Universal Robots PolyScope program: DEMO_ghost4.urp

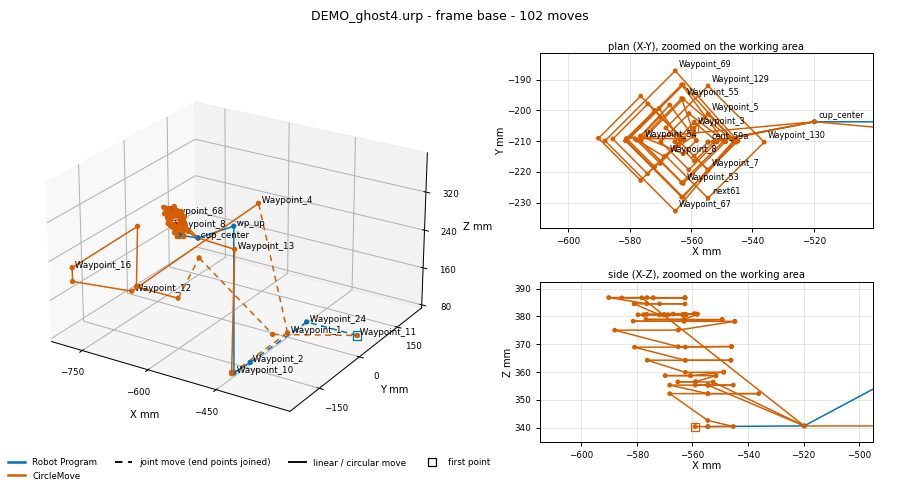
[picture p0: tool path of DEMO_ghost4.urp in frame base, 102 of 102 moves have a stored position in this frame; points joined in program order, loops and branches not executed]
Program DEMO_ghost4 (createdIn=3.3.3.292 lastSavedIn=3.3.3.292 directory=/programs/usbdisk_0 installation=default robotSerialNumber=2016353566)
Calibrated DH parameters: a=[0.000241, -0.028217, -0.285075, -0.000076, 0.000104, 0]; d=[0.089155, 574.834368, -342.811798, -231.912434, 0.094822, 0.082605]; alpha=[1.570306, 0.000738, 0.001161, 1.569845, -1.570892, 0]; deltaTheta=[0.000027, 1.504353, -0.747309, -0.757122, 0.000051, -0.000036]
Robot Program (runOnlyOnce=true motionType=MoveJ speed=1.047198 acceleration=1.396263 recalculateMotions=false)
  'c250g_w360g'
  URCap com.ur.urcap.OnRobot.HelloWorldNode data=depthCompensate = false
    | width = 40
    | name = RG2(40)
    | force = 40
  MoveJ speed 20 deg/s, acceleration 30 deg/s^2 (recalculateMotions=false)
    Waypoint Waypoint_11: TCP in base x=-315.829 y=31.141 z=99.108 mm, rx=0.0221 ry=-2.2156 rz=2.1951 rad; joints [-58.8, -68.323, 115.476, -47.806, -58.377, -1.11] deg; flange x=-314.66 y=223.315 z=100.907 mm, rx=1.5801 ry=0.0158 rz=-0.0251 rad
    Waypoint Waypoint_24: TCP in base x=-426.481 y=31.172 z=99.122 mm, rx=0.0223 ry=-2.2158 rz=2.195 rad; joints [-47.924, -59.45, 100.701, -42.012, -47.495, -0.947] deg; flange x=-425.323 y=223.315 z=100.907 mm, rx=1.5801 ry=0.0158 rz=-0.0251 rad
    Waypoint Waypoint_2: TCP in base x=-433.696 y=-162.819 z=93.941 mm, rx=0.4331 ry=2.0006 rz=-1.9847 rad; joints [-28.835, -67.033, 114.523, -48.696, -28.414, 25.171] deg; flange x=-432.521 y=29.34 z=95.724 mm, rx=1.5534 ry=-0.3363 rz=0.3238 rad
  MoveL speed 76.2 mm/s, acceleration 1198.88 mm/s^2 (recalculateMotions=false) feature=Base
    Waypoint Waypoint_10: TCP in base x=-443.417 y=-203.708 z=87.403 mm, rx=0.7795 ry=1.7327 rz=-1.7213 rad; joints [-23.409, -66.24, 114.647, -49.886, -22.989, 49.486] deg; flange x=-442.26 y=-11.553 z=89.193 mm, rx=1.4755 ry=-0.6639 rz=0.6489 rad
  URCap com.ur.urcap.OnRobot.HelloWorldNode data=depthCompensate = false
    | width = 0
    | name = RG2(0)
    | force = 40
  MoveL speed 76.2 mm/s, acceleration 254 mm/s^2 (recalculateMotions=false) feature=Base
    Waypoint wp_up: TCP in base x=-443.405 y=-203.725 z=381.397 mm, rx=0.7794 ry=1.7329 rz=-1.7213 rad; joints [-23.396, -84.47, 89.34, -6.233, -23.004, 49.36] deg; flange x=-442.26 y=-11.553 z=383.168 mm, rx=1.4755 ry=-0.6639 rz=0.6489 rad
    Waypoint cup_center: TCP in base x=-519.8 y=-203.671 z=340.608 mm, rx=0.7796 ry=1.7328 rz=-1.7213 rad; joints [-19.983, -73.438, 82.009, -10.178, -19.586, 49.619] deg; flange x=-518.65 y=-11.524 z=342.376 mm, rx=1.4756 ry=-0.6638 rz=0.6489 rad
    Waypoint cent_59a: motionParameters(jointSpeed=1.047198 jointAcceleration=1.396263 cartesianSpeed=0.0254 cartesianAcceleration=0.0508 blendRadius=0); TCP in base x=-554.479 y=-210.348 z=340.374 mm, rx=0.8933 ry=1.6233 rz=-1.6133 rad; joints [-18.076, -68.796, 75.751, -8.732, -17.687, 59.013] deg; flange x=-553.37 y=-18.19 z=342.205 mm, rx=1.432 ry=-0.788 rz=0.7724 rad
  MoveP speed 17.78 mm/s, acceleration 10.16 mm/s^2 (blendRadius=0.00762 recalculateMotions=false) feature=Base
    CircleMove
      Waypoint Waypoint_3: TCP in base x=-559.014 y=-205.731 z=340.364 mm, rx=0.8959 ry=1.6205 rz=-1.6105 rad; joints [-18.383, -68.07, 74.735, -8.411, -17.996, 59.2] deg; flange x=-557.938 y=-13.596 z=342.198 mm, rx=1.4308 ry=-0.7909 rz=0.7754 rad
      Waypoint Waypoint_5: TCP in base x=-554.401 y=-201.21 z=340.352 mm, rx=0.897 ry=1.6193 rz=-1.6092 rad; joints [-18.99, -68.615, 75.506, -8.574, -18.608, 59.25] deg; flange x=-553.342 y=-9.005 z=342.152 mm, rx=1.4302 ry=-0.7924 rz=0.777 rad
    CircleMove
      Waypoint Waypoint_6: TCP in base x=-545.287 y=-210.272 z=340.388 mm, rx=0.8993 ry=1.617 rz=-1.607 rad; joints [-18.381, -70.062, 77.509, -9.19, -18.007, 59.5] deg; flange x=-544.195 y=-18.156 z=342.164 mm, rx=1.4293 ry=-0.7948 rz=0.7796 rad
      Waypoint Waypoint_7: TCP in base x=-554.475 y=-219.387 z=342.569 mm, rx=0.9035 ry=1.6129 rz=-1.6029 rad; joints [-17.172, -68.988, 75.704, -8.585, -16.788, 59.988] deg; flange x=-553.372 y=-27.212 z=344.349 mm, rx=1.4274 ry=-0.7997 rz=0.7842 rad
    '0.54start'
    CircleMove
      Waypoint Waypoint_128: TCP in base x=-568.169 y=-205.675 z=352.208 mm, rx=0.9085 ry=1.6076 rz=-1.598 rad; joints [-18.096, -66.938, 71.401, -6.222, -17.71, 60.295] deg; flange x=-567.062 y=-13.525 z=353.986 mm, rx=1.4251 ry=-0.8054 rz=0.7898 rad
      Waypoint Waypoint_129: motionParameters(blendRadius=0.004); TCP in base x=-554.437 y=-191.989 z=352.215 mm, rx=0.9129 ry=1.6031 rz=-1.5935 rad; joints [-19.903, -68.595, 73.735, -6.737, -19.508, 60.5] deg; flange x=-553.301 y=0.226 z=354.016 mm, rx=1.423 ry=-0.8105 rz=0.7947 rad
    CircleMove
      Waypoint Waypoint_130: TCP in base x=-536.157 y=-210.292 z=352.228 mm, rx=0.915 ry=1.6009 rz=-1.5913 rad; joints [-18.704, -71.524, 77.755, -7.932, -18.312, 60.8] deg; flange x=-535.028 y=-18.073 z=353.996 mm, rx=1.422 ry=-0.813 rz=0.7972 rad
      Waypoint next61: motionParameters(blendRadius=0.005994); TCP in base x=-554.45 y=-228.557 z=352.204 mm, rx=0.9153 ry=1.6006 rz=-1.5912 rad; joints [-16.246, -69.278, 74.691, -7.369, -15.857, 61.065] deg; flange x=-553.316 y=-36.41 z=353.989 mm, rx=1.4221 ry=-0.813 rz=0.7972 rad
    CircleMove
      Waypoint Waypoint_8: TCP in base x=-568.176 y=-214.818 z=355.297 mm, rx=0.9193 ry=1.5964 rz=-1.5871 rad; joints [-17.207, -67.147, 71.244, -5.939, -16.808, 61.299] deg; flange x=-567.033 y=-22.648 z=357.097 mm, rx=1.4201 ry=-0.8178 rz=0.8018 rad
      Waypoint Waypoint_9: motionParameters(blendRadius=0.00635); TCP in base x=-554.434 y=-201.143 z=355.277 mm, rx=0.9216 ry=1.5938 rz=-1.5844 rad; joints [-18.997, -68.829, 73.615, -6.45, -18.604, 61.33] deg; flange x=-553.312 y=-8.943 z=357.064 mm, rx=1.4189 ry=-0.8206 rz=0.8048 rad
    CircleMove
      Waypoint Waypoint_14: motionParameters(blendRadius=0); TCP in base x=-545.305 y=-210.255 z=355.292 mm, rx=0.9229 ry=1.5926 rz=-1.5832 rad; joints [-18.387, -70.291, 75.635, -7.064, -18.002, 61.5] deg; flange x=-544.181 y=-18.11 z=357.05 mm, rx=1.4184 ry=-0.822 rz=0.8064 rad
      Waypoint Waypoint_20: motionParameters(blendRadius=0.005); TCP in base x=-554.453 y=-219.368 z=355.292 mm, rx=0.9273 ry=1.5881 rz=-1.5788 rad; joints [-17.169, -69.172, 74.091, -6.77, -16.781, 62] deg; flange x=-553.328 y=-27.252 z=357.074 mm, rx=1.4165 ry=-0.827 rz=0.8112 rad
    CircleMove
      Waypoint Waypoint_23: motionParameters(jointSpeed=1.047198 jointAcceleration=1.396263 cartesianSpeed=0.00508 cartesianAcceleration=0.00508 blendRadius=0); TCP in base x=-558.979 y=-214.836 z=355.315 mm, rx=0.9277 ry=1.5875 rz=-1.5783 rad; joints [-17.487, -68.448, 73.084, -6.446, -17.093, 62] deg; flange x=-557.885 y=-22.655 z=357.065 mm, rx=1.4161 ry=-0.8276 rz=0.8116 rad
      Waypoint Waypoint_26: motionParameters(jointSpeed=1.047198 jointAcceleration=1.396263 cartesianSpeed=0.00508 cartesianAcceleration=0.00508 blendRadius=0); TCP in base x=-554.401 y=-210.229 z=355.266 mm, rx=0.9283 ry=1.5869 rz=-1.5775 rad; joints [-18.089, -69.016, 73.873, -6.61, -17.699, 62] deg; flange x=-553.278 y=-18.086 z=357.079 mm, rx=1.4159 ry=-0.8284 rz=0.8125 rad
  Wait Sleep waitTime=0.5
  'bloom finished'
  MoveL speed 76.2 mm/s, acceleration 635 mm/s^2 (recalculateMotions=false) feature=Base
    Waypoint cup_cent: TCP in base x=-519.766 y=-203.654 z=340.589 mm, rx=0.7795 ry=1.7327 rz=-1.7212 rad; joints [-19.983, -73.438, 82.009, -10.178, -19.586, 49.619] deg; flange x=-518.65 y=-11.524 z=342.376 mm, rx=1.4756 ry=-0.6638 rz=0.6489 rad
  Wait Sleep waitTime=30
  'first_pour'
  MoveP speed 20.32 mm/s, acceleration 10.16 mm/s^2 (blendRadius=0.00762 recalculateMotions=false) feature=Base
    Waypoint cent_63a: TCP in base x=-552.569 y=-210.233 z=356.4 mm, rx=0.941 ry=1.5723 rz=-1.5646 rad; joints [-18.152, -69.253, 74.075, -6.42, -17.753, 62.988] deg; flange x=-551.431 y=-18.061 z=358.005 mm, rx=1.4088 ry=-0.8432 rz=0.8277 rad
    Loop Counting (count=2) loopVariable(name=Loop_1)
      MoveP speed 25.4 mm/s, acceleration 7.62 mm/s^2 (blendRadius=0.000991 recalculateMotions=false) feature=Base
        CircleMove
          Waypoint Waypoint_43: TCP in base x=-558.846 y=-216.512 z=356.423 mm, rx=0.9408 ry=1.5725 rz=-1.5645 rad; joints [-17.321, -68.472, 72.982, -6.192, -16.918, 63.063] deg; flange x=-557.773 y=-24.37 z=358.046 mm, rx=1.4089 ry=-0.8431 rz=0.8275 rad
          Waypoint Waypoint_44: motionParameters(blendRadius=0.001); TCP in base x=-565.247 y=-210.188 z=356.452 mm, rx=0.9411 ry=1.5723 rz=-1.5646 rad; joints [-17.754, -67.459, 71.547, -5.734, -17.346, 63.022] deg; flange x=-564.107 y=-17.986 z=358.106 mm, rx=1.4089 ry=-0.8432 rz=0.8274 rad
        CircleMove
          Waypoint Waypoint_45: TCP in base x=-558.906 y=-203.746 z=356.509 mm, rx=0.941 ry=1.5725 rz=-1.5648 rad; joints [-18.59, -68.241, 72.647, -5.977, -18.179, 62.947] deg; flange x=-557.747 y=-11.574 z=358.115 mm, rx=1.4089 ry=-0.8432 rz=0.8274 rad
          Waypoint next_64a: motionParameters(jointSpeed=1.047198 jointAcceleration=1.396263 cartesianSpeed=0.01778 cartesianAcceleration=0.0254); TCP in base x=-551.565 y=-210.182 z=358.675 mm, rx=0.9523 ry=1.5601 rz=-1.5525 rad; joints [-18.186, -69.425, 73.976, -6.162, -17.791, 63.995] deg; flange x=-550.42 y=-18.05 z=360.298 mm, rx=1.4034 ry=-0.8565 rz=0.841 rad
    Waypoint cent_64a: TCP in base x=-551.561 y=-210.22 z=358.653 mm, rx=0.9522 ry=1.5602 rz=-1.5524 rad; joints [-18.188, -69.428, 73.979, -6.156, -17.787, 63.996] deg; flange x=-550.399 y=-18.042 z=360.305 mm, rx=1.4033 ry=-0.8567 rz=0.841 rad
    Loop Counting (count=2) loopVariable(name=Loop_4)
      MoveP speed 25.4 mm/s, acceleration 7.62 mm/s^2 (blendRadius=0.0127 recalculateMotions=false) feature=Base
        CircleMove
          Waypoint Waypoint_46: TCP in base x=-560.706 y=-219.295 z=358.709 mm, rx=0.9523 ry=1.5602 rz=-1.5526 rad; joints [-16.988, -68.293, 72.397, -5.828, -16.59, 64.115] deg; flange x=-559.547 y=-27.161 z=360.32 mm, rx=1.4033 ry=-0.8566 rz=0.841 rad
          Waypoint Waypoint_47: TCP in base x=-569.84 y=-210.183 z=358.713 mm, rx=0.9541 ry=1.5583 rz=-1.5508 rad; joints [-17.613, -66.823, 70.313, -5.154, -17.206, 64.2] deg; flange x=-568.694 y=-17.975 z=360.351 mm, rx=1.4024 ry=-0.8587 rz=0.8428 rad
        CircleMove
          Waypoint Waypoint_48: TCP in base x=-560.679 y=-200.996 z=358.67 mm, rx=0.9586 ry=1.5532 rz=-1.5457 rad; joints [-18.803, -67.956, 71.92, -5.521, -18.397, 64.5] deg; flange x=-559.514 y=-8.81 z=360.343 mm, rx=1.4001 ry=-0.8642 rz=0.8483 rad
          Waypoint Waypoint_49: TCP in base x=-548.75 y=-210.183 z=359.952 mm, rx=0.9634 ry=1.5478 rz=-1.5403 rad; joints [-18.284, -69.828, 74.343, -6.105, -17.888, 64.987] deg; flange x=-547.634 y=-17.997 z=361.584 mm, rx=1.3975 ry=-0.87 rz=0.8544 rad
    Waypoint cent_65a: TCP in base x=-548.775 y=-210.166 z=359.952 mm, rx=0.9635 ry=1.5477 rz=-1.5403 rad; joints [-18.285, -69.83, 74.341, -6.112, -17.89, 64.989] deg; flange x=-547.641 y=-17.982 z=361.615 mm, rx=1.3976 ry=-0.87 rz=0.8543 rad
    Loop Counting (count=2) loopVariable(name=Loop_5)
      MoveP speed 25.4 mm/s, acceleration 7.62 mm/s^2 (blendRadius=0.00889 recalculateMotions=false) feature=Base
        CircleMove
          Waypoint Waypoint_53: motionParameters(blendRadius=0.01); TCP in base x=-562.543 y=-223.776 z=359.879 mm, rx=0.9638 ry=1.5475 rz=-1.5404 rad; joints [-16.485, -68.115, 71.969, -5.613, -16.087, 65.165] deg; flange x=-561.352 y=-31.679 z=361.549 mm, rx=1.3975 ry=-0.8701 rz=0.8544 rad
          Waypoint Waypoint_54: motionParameters(blendRadius=0.001); TCP in base x=-576.264 y=-210.006 z=364.262 mm, rx=0.9665 ry=1.5445 rz=-1.5375 rad; joints [-17.428, -65.93, 68.223, -3.945, -17.019, 65.298] deg; flange x=-575.07 y=-17.878 z=365.892 mm, rx=1.396 ry=-0.8734 rz=0.8575 rad
        CircleMove
          Waypoint Waypoint_55: motionParameters(blendRadius=0.017); TCP in base x=-562.564 y=-196.291 z=364.226 mm, rx=0.9682 ry=1.5427 rz=-1.5356 rad; joints [-19.197, -67.636, 70.663, -4.527, -18.788, 65.3] deg; flange x=-561.358 y=-4.147 z=365.85 mm, rx=1.395 ry=-0.8756 rz=0.8597 rad
          Waypoint Waypoint_56: TCP in base x=-546.154 y=-210.035 z=364.248 mm, rx=0.9748 ry=1.5354 rz=-1.5282 rad; joints [-18.388, -70.245, 74.289, -5.631, -17.982, 65.989] deg; flange x=-545 y=-17.838 z=365.849 mm, rx=1.3916 ry=-0.8836 rz=0.8676 rad
    Waypoint cent_66a: TCP in base x=-546.18 y=-209.995 z=364.224 mm, rx=0.9749 ry=1.5354 rz=-1.5283 rad; joints [-18.388, -70.245, 74.289, -5.631, -17.982, 65.989] deg; flange x=-545 y=-17.838 z=365.849 mm, rx=1.3916 ry=-0.8836 rz=0.8676 rad
    Loop Counting (count=1) loopVariable(name=Loop_6)
      MoveP speed 20.32 mm/s, acceleration 12.7 mm/s^2 (blendRadius=0.00762 recalculateMotions=false) feature=Base
        CircleMove
          Waypoint Waypoint_60: motionParameters(blendRadius=0.017); TCP in base x=-562.588 y=-228.258 z=364.234 mm, rx=0.9752 ry=1.5351 rz=-1.5282 rad; joints [-16.04, -68.219, 71.487, -5.08, -15.637, 66.248] deg; flange x=-561.379 y=-36.137 z=365.834 mm, rx=1.3915 ry=-0.8839 rz=0.868 rad
          Waypoint Waypoint_61: motionParameters(blendRadius=0.007); TCP in base x=-580.842 y=-209.916 z=368.929 mm, rx=0.9773 ry=1.5327 rz=-1.5258 rad; joints [-17.299, -65.283, 66.601, -3, -16.889, 66.298] deg; flange x=-579.639 y=-17.803 z=370.568 mm, rx=1.3904 ry=-0.8864 rz=0.8704 rad
        CircleMove
          Waypoint Waypoint_62: motionParameters(blendRadius=0.017); TCP in base x=-562.548 y=-191.661 z=368.972 mm, rx=0.9795 ry=1.5303 rz=-1.5233 rad; joints [-19.652, -67.569, 69.875, -3.788, -19.239, 66.3] deg; flange x=-561.345 y=0.528 z=370.583 mm, rx=1.3891 ry=-0.8893 rz=0.8731 rad
          Waypoint Waypoint_63: TCP in base x=-545.944 y=-209.955 z=369.156 mm, rx=0.986 ry=1.523 rz=-1.5159 rad; joints [-18.4, -70.325, 73.675, -4.956, -17.998, 67.012] deg; flange x=-544.772 y=-17.793 z=370.78 mm, rx=1.3858 ry=-0.897 rz=0.8809 rad
    Waypoint cent_67a: motionParameters(blendRadius=0); TCP in base x=-545.939 y=-209.974 z=369.159 mm, rx=0.9859 ry=1.5231 rz=-1.516 rad; joints [-18.4, -70.325, 73.675, -4.956, -17.998, 67.012] deg; flange x=-544.772 y=-17.793 z=370.78 mm, rx=1.3858 ry=-0.897 rz=0.8809 rad
    Loop Counting (count=1) loopVariable(name=Loop_7)
      MoveP speed 25.4 mm/s, acceleration 15.24 mm/s^2 (blendRadius=0.0127 recalculateMotions=false) feature=Base
        CircleMove
          Waypoint Waypoint_67: TCP in base x=-565.085 y=-232.781 z=369.094 mm, rx=0.986 ry=1.523 rz=-1.5159 rad; joints [-15.52, -67.963, 70.407, -4.342, -15.115, 67.319] deg; flange x=-563.888 y=-40.649 z=370.752 mm, rx=1.3858 ry=-0.8971 rz=0.8809 rad
          Waypoint Waypoint_68: TCP in base x=-587.967 y=-209.866 z=375.056 mm, rx=0.986 ry=1.523 rz=-1.516 rad; joints [-17.093, -64.232, 64.164, -1.646, -16.685, 67.133] deg; flange x=-586.76 y=-17.77 z=376.722 mm, rx=1.3857 ry=-0.8971 rz=0.881 rad
        CircleMove
          Waypoint Waypoint_69: TCP in base x=-565.128 y=-187.05 z=375.084 mm, rx=0.9906 ry=1.5178 rz=-1.5108 rad; joints [-20.007, -67.119, 68.337, -2.69, -19.596, 67.3] deg; flange x=-563.912 y=5.13 z=376.733 mm, rx=1.3832 ry=-0.9028 rz=0.8865 rad
          Waypoint Waypoint_70: TCP in base x=-544.745 y=-209.896 z=378.224 mm, rx=0.9966 ry=1.511 rz=-1.5039 rad; joints [-18.446, -70.561, 72.659, -3.709, -18.038, 67.995] deg; flange x=-543.561 y=-17.743 z=379.926 mm, rx=1.38 ry=-0.9102 rz=0.8937 rad
    Waypoint cent_68a: motionParameters(blendRadius=0); TCP in base x=-544.738 y=-209.887 z=378.224 mm, rx=0.9967 ry=1.5109 rz=-1.5039 rad; joints [-18.446, -70.561, 72.659, -3.709, -18.038, 67.995] deg; flange x=-543.561 y=-17.743 z=379.926 mm, rx=1.38 ry=-0.9102 rz=0.8937 rad
    Loop Counting (count=1) loopVariable(name=Loop_8)
      MoveP speed 20.32 mm/s, acceleration 10.16 mm/s^2 (blendRadius=0.01778 recalculateMotions=false) feature=Base
        CircleMove
          Waypoint Waypoint_74: TCP in base x=-563.018 y=-228.234 z=378.278 mm, rx=0.9965 ry=1.5111 rz=-1.504 rad; joints [-16.037, -68.237, 69.448, -3.066, -15.632, 68.245] deg; flange x=-561.863 y=-36.038 z=379.938 mm, rx=1.3801 ry=-0.9101 rz=0.8937 rad
          Waypoint Waypoint_75: TCP in base x=-581.336 y=-209.872 z=378.296 mm, rx=0.9987 ry=1.5086 rz=-1.5017 rad; joints [-17.287, -65.231, 65.151, -1.641, -16.881, 68.3] deg; flange x=-580.145 y=-17.767 z=379.96 mm, rx=1.3789 ry=-0.9127 rz=0.8963 rad
        CircleMove
          Waypoint Waypoint_76: TCP in base x=-563.043 y=-191.607 z=378.299 mm, rx=1.001 ry=1.5061 rz=-1.499 rad; joints [-19.639, -67.543, 68.46, -2.435, -19.231, 68.3] deg; flange x=-561.838 y=0.575 z=379.991 mm, rx=1.3776 ry=-0.9155 rz=0.8991 rad
          Waypoint Waypoint_77: TCP in base x=-549.329 y=-209.898 z=378.857 mm, rx=1.0072 ry=1.4988 rz=-1.4919 rad; joints [-18.294, -69.911, 71.674, -3.397, -17.89, 69.001] deg; flange x=-548.141 y=-17.731 z=380.578 mm, rx=1.3741 ry=-0.9232 rz=0.9068 rad
    Waypoint cent_69a: motionParameters(blendRadius=0); TCP in base x=-549.318 y=-209.9 z=378.893 mm, rx=1.0071 ry=1.4989 rz=-1.4919 rad; joints [-18.295, -69.91, 71.672, -3.397, -17.889, 69] deg; flange x=-548.152 y=-17.715 z=380.586 mm, rx=1.3741 ry=-0.9232 rz=0.9067 rad
    Loop Counting (count=2) loopVariable(name=Loop_9)
      MoveP speed 25.4 mm/s, acceleration 15.24 mm/s^2 (blendRadius=0.01524 recalculateMotions=false) feature=Base
        CircleMove
          Waypoint Waypoint_81: TCP in base x=-563.047 y=-223.508 z=378.892 mm, rx=1.0071 ry=1.4991 rz=-1.4922 rad; joints [-16.502, -68.178, 69.266, -2.9, -16.096, 69.183] deg; flange x=-561.809 y=-31.374 z=380.607 mm, rx=1.3741 ry=-0.9232 rz=0.9067 rad
          Waypoint Waypoint_82: TCP in base x=-576.75 y=-209.782 z=378.943 mm, rx=1.0085 ry=1.4974 rz=-1.4906 rad; joints [-17.435, -65.916, 66.045, -1.846, -17.021, 69.2] deg; flange x=-575.569 y=-17.65 z=380.628 mm, rx=1.3733 ry=-0.9248 rz=0.9081 rad
        CircleMove
          Waypoint Waypoint_83: TCP in base x=-563.039 y=-196.086 z=378.956 mm, rx=1.0113 ry=1.4943 rz=-1.4875 rad; joints [-19.205, -67.653, 68.522, -2.427, -18.79, 69.3] deg; flange x=-561.816 y=-3.9 z=380.628 mm, rx=1.3717 ry=-0.9284 rz=0.9117 rad
          Waypoint Waypoint_84: TCP in base x=-558.279 y=-209.805 z=380.853 mm, rx=1.0176 ry=1.4869 rz=-1.4801 rad; joints [-18.012, -68.634, 69.62, -2.656, -17.596, 70.014] deg; flange x=-557.077 y=-17.641 z=382.537 mm, rx=1.368 ry=-0.9363 rz=0.9195 rad
    Waypoint cent_70a: motionParameters(blendRadius=0); TCP in base x=-558.292 y=-209.819 z=380.817 mm, rx=1.0176 ry=1.4868 rz=-1.48 rad; joints [-18.012, -68.634, 69.62, -2.656, -17.596, 70.014] deg; flange x=-557.077 y=-17.641 z=382.537 mm, rx=1.368 ry=-0.9363 rz=0.9195 rad
    Loop Counting (count=2) loopVariable(name=Loop_10)
      MoveP speed 25.4 mm/s, acceleration 7.62 mm/s^2 (blendRadius=0.01524 recalculateMotions=false) feature=Base
        CircleMove
          Waypoint Waypoint_88: TCP in base x=-562.522 y=-214.098 z=380.823 mm, rx=1.0174 ry=1.4871 rz=-1.4802 rad; joints [-17.45, -68.086, 68.86, -2.491, -17.044, 70.072] deg; flange x=-561.375 y=-21.945 z=382.497 mm, rx=1.368 ry=-0.9363 rz=0.9197 rad
          Waypoint Waypoint_89: TCP in base x=-576.448 y=-208.299 z=380.755 mm, rx=1.0178 ry=1.4866 rz=-1.48 rad; joints [-17.594, -65.943, 65.81, -1.566, -17.185, 70.057] deg; flange x=-575.176 y=-16.127 z=382.499 mm, rx=1.368 ry=-0.9364 rz=0.9198 rad
        CircleMove
          Waypoint Waypoint_90: TCP in base x=-566.936 y=-198.208 z=380.882 mm, rx=1.0178 ry=1.4864 rz=-1.4797 rad; joints [-18.862, -67.122, 67.491, -1.955, -18.454, 69.942] deg; flange x=-565.787 y=-6.072 z=382.545 mm, rx=1.3679 ry=-0.9364 rz=0.9198 rad
          Waypoint Waypoint_91: TCP in base x=-559.322 y=-208.319 z=380.954 mm, rx=1.0232 ry=1.4802 rz=-1.4738 rad; joints [-18.124, -68.45, 69.353, -2.545, -17.712, 70.51] deg; flange x=-558.115 y=-16.17 z=382.618 mm, rx=1.3647 ry=-0.9432 rz=0.9265 rad
    Waypoint cent_71a: TCP in base x=-559.302 y=-208.361 z=380.931 mm, rx=1.0231 ry=1.4802 rz=-1.4737 rad; joints [-18.124, -68.45, 69.353, -2.545, -17.712, 70.51] deg; flange x=-558.115 y=-16.17 z=382.618 mm, rx=1.3647 ry=-0.9432 rz=0.9265 rad
    Loop Counting (count=2) loopVariable(name=Loop_12)
      MoveP speed 25.4 mm/s, acceleration 12.7 mm/s^2 (blendRadius=0.009144 recalculateMotions=false) feature=Base
        CircleMove
          Waypoint Waypoint_102: TCP in base x=-568.74 y=-214.984 z=380.648 mm, rx=1.0282 ry=1.4742 rz=-1.4677 rad; joints [-17.172, -67.201, 67.633, -2.158, -16.762, 71.096] deg; flange x=-567.503 y=-22.871 z=382.349 mm, rx=1.3615 ry=-0.9497 rz=0.9331 rad
          Waypoint Waypoint_103: TCP in base x=-579.589 y=-208.445 z=380.607 mm, rx=1.0284 ry=1.474 rz=-1.4678 rad; joints [-17.484, -65.482, 65.163, -1.377, -17.066, 71.063] deg; flange x=-578.28 y=-16.295 z=382.372 mm, rx=1.3615 ry=-0.9498 rz=0.933 rad
        CircleMove
          Waypoint Waypoint_104: TCP in base x=-570.405 y=-199.334 z=380.61 mm, rx=1.0284 ry=1.474 rz=-1.4678 rad; joints [-18.647, -66.643, 66.855, -1.784, -18.218, 70.948] deg; flange x=-569.182 y=-7.153 z=382.234 mm, rx=1.3612 ry=-0.95 rz=0.933 rad
          Waypoint Waypoint_105: TCP in base x=-563.455 y=-209.727 z=380.664 mm, rx=1.0332 ry=1.4682 rz=-1.462 rad; joints [-17.856, -67.871, 68.586, -2.37, -17.44, 71.5] deg; flange x=-562.255 y=-17.545 z=382.308 mm, rx=1.3584 ry=-0.9561 rz=0.9393 rad
    Waypoint cent_72a: TCP in base x=-563.47 y=-209.73 z=380.649 mm, rx=1.0333 ry=1.468 rz=-1.4618 rad; joints [-17.856, -67.871, 68.586, -2.37, -17.44, 71.5] deg; flange x=-562.255 y=-17.545 z=382.308 mm, rx=1.3584 ry=-0.9561 rz=0.9393 rad
    Loop Counting (count=2) loopVariable(name=Loop_13)
      MoveP speed 25.4 mm/s, acceleration 7.62 mm/s^2 (blendRadius=0.00762 recalculateMotions=false) feature=Base
        CircleMove
          Waypoint Waypoint_109: TCP in base x=-570.008 y=-217.238 z=380.618 mm, rx=1.0381 ry=1.4623 rz=-1.4557 rad; joints [-16.911, -67.046, 67.415, -2.151, -16.51, 72.099] deg; flange x=-568.864 y=-25.114 z=382.324 mm, rx=1.3557 ry=-0.9623 rz=0.9456 rad
          Waypoint Waypoint_110: TCP in base x=-577.609 y=-209.707 z=380.617 mm, rx=1.038 ry=1.4625 rz=-1.4557 rad; joints [-17.426, -65.778, 65.598, -1.546, -17.025, 72.046] deg; flange x=-576.464 y=-17.46 z=382.32 mm, rx=1.3557 ry=-0.9623 rz=0.9457 rad
        CircleMove
          Waypoint Waypoint_111: TCP in base x=-570.059 y=-202.078 z=380.601 mm, rx=1.0382 ry=1.4621 rz=-1.4556 rad; joints [-18.391, -66.748, 66.993, -1.877, -17.989, 71.954] deg; flange x=-568.886 y=-9.896 z=382.306 mm, rx=1.3556 ry=-0.9624 rz=0.9458 rad
          Waypoint Waypoint_112: TCP in base x=-562.307 y=-209.55 z=380.601 mm, rx=1.0435 ry=1.4559 rz=-1.4495 rad; joints [-17.906, -68.038, 68.819, -2.457, -17.498, 72.5] deg; flange x=-561.122 y=-17.397 z=382.318 mm, rx=1.3523 ry=-0.9691 rz=0.9523 rad
    Waypoint cent_73a: TCP in base x=-562.311 y=-209.571 z=380.637 mm, rx=1.0433 ry=1.456 rz=-1.4496 rad; joints [-17.906, -68.038, 68.819, -2.457, -17.498, 72.5] deg; flange x=-561.122 y=-17.397 z=382.318 mm, rx=1.3523 ry=-0.9691 rz=0.9523 rad
    Loop Counting (count=2) loopVariable(name=Loop_2)
      MoveP speed 25.4 mm/s, acceleration 12.7 mm/s^2 (blendRadius=0.0127 recalculateMotions=false) feature=Base
        CircleMove
          Waypoint Waypoint_27: TCP in base x=-571.824 y=-218.312 z=380.589 mm, rx=1.0468 ry=1.4519 rz=-1.446 rad; joints [-16.76, -66.807, 67.086, -2.058, -16.338, 72.92] deg; flange x=-570.604 y=-26.146 z=382.249 mm, rx=1.3501 ry=-0.9733 rz=0.9562 rad
          Waypoint Waypoint_28: TCP in base x=-581.001 y=-209.12 z=384.522 mm, rx=1.0504 ry=1.4476 rz=-1.4417 rad; joints [-17.372, -65.273, 64.295, -0.732, -16.95, 73.198] deg; flange x=-579.732 y=-17.013 z=386.239 mm, rx=1.3478 ry=-0.9779 rz=0.9608 rad
        CircleMove
          Waypoint Waypoint_29: TCP in base x=-571.869 y=-199.996 z=384.529 mm, rx=1.0537 ry=1.4434 rz=-1.4378 rad; joints [-18.539, -66.453, 65.998, -1.148, -18.114, 73.4] deg; flange x=-570.582 y=-7.804 z=386.232 mm, rx=1.3458 ry=-0.9821 rz=0.9649 rad
          Waypoint Waypoint_30: TCP in base x=-562.691 y=-209.079 z=384.506 mm, rx=1.054 ry=1.443 rz=-1.4372 rad; joints [-17.941, -67.986, 68.177, -1.842, -17.523, 73.5] deg; flange x=-561.432 y=-16.948 z=386.217 mm, rx=1.3455 ry=-0.9827 rz=0.9656 rad
    Loop Counting (count=2) loopVariable(name=Loop_11)
      MoveP speed 25.4 mm/s, acceleration 12.7 mm/s^2 (blendRadius=0.00762 recalculateMotions=false) feature=Base
        CircleMove
          Waypoint Waypoint_31: TCP in base x=-576.39 y=-222.782 z=384.564 mm, rx=1.0542 ry=1.4429 rz=-1.4372 rad; joints [-16.192, -66.201, 65.641, -1.273, -15.77, 73.687] deg; flange x=-575.167 y=-30.631 z=386.213 mm, rx=1.3455 ry=-0.9827 rz=0.9655 rad
          Waypoint Waypoint_32: TCP in base x=-590.123 y=-209.046 z=386.805 mm, rx=1.0541 ry=1.4429 rz=-1.4373 rad; joints [-17.116, -63.875, 61.913, 0.227, -16.685, 73.584] deg; flange x=-588.856 y=-16.902 z=388.52 mm, rx=1.3454 ry=-0.9828 rz=0.9654 rad
        CircleMove
          Waypoint Waypoint_33: TCP in base x=-576.378 y=-195.306 z=386.779 mm, rx=1.0589 ry=1.4369 rz=-1.4312 rad; joints [-18.839, -65.663, 64.537, -0.44, -18.413, 73.9] deg; flange x=-575.135 y=-3.136 z=388.449 mm, rx=1.3422 ry=-0.9892 rz=0.972 rad
          Waypoint Waypoint_34: TCP in base x=-562.714 y=-209.2 z=386.73 mm, rx=1.0613 ry=1.4341 rz=-1.4286 rad; joints [-17.933, -67.991, 67.859, -1.517, -17.505, 74.2] deg; flange x=-561.422 y=-17.034 z=388.441 mm, rx=1.3407 ry=-0.9921 rz=0.9747 rad
    Waypoint cent_74a: TCP in base x=-562.697 y=-209.216 z=386.762 mm, rx=1.0612 ry=1.4342 rz=-1.4287 rad; joints [-17.933, -67.991, 67.859, -1.517, -17.505, 74.2] deg; flange x=-561.422 y=-17.034 z=388.441 mm, rx=1.3407 ry=-0.9921 rz=0.9747 rad
    Loop Counting (count=2) loopVariable(name=Loop_3)
      MoveP speed 15.24 mm/s, acceleration 12.7 mm/s^2 (blendRadius=0.01524 recalculateMotions=false) feature=Base
        CircleMove
          Waypoint Waypoint_35: TCP in base x=-574.136 y=-220.623 z=386.706 mm, rx=1.0613 ry=1.4339 rz=-1.4286 rad; joints [-16.468, -66.502, 65.754, -1.04, -16.045, 74.354] deg; flange x=-572.863 y=-28.469 z=388.397 mm, rx=1.3407 ry=-0.9921 rz=0.9749 rad
          Waypoint Waypoint_36: TCP in base x=-585.437 y=-209.266 z=386.693 mm, rx=1.061 ry=1.434 rz=-1.4282 rad; joints [-17.235, -64.57, 62.963, -0.089, -16.815, 74.269] deg; flange x=-584.283 y=-17.044 z=388.341 mm, rx=1.3406 ry=-0.9921 rz=0.9751 rad
        CircleMove
          Waypoint Waypoint_37: TCP in base x=-574.045 y=-197.86 z=386.641 mm, rx=1.061 ry=1.4339 rz=-1.4282 rad; joints [-18.672, -66.062, 65.128, -0.629, -18.261, 74.13] deg; flange x=-572.805 y=-5.668 z=388.349 mm, rx=1.3407 ry=-0.992 rz=0.9753 rad
          Waypoint Waypoint_38: motionParameters(jointSpeed=1.047198 jointAcceleration=1.396263 cartesianSpeed=0.0127 cartesianAcceleration=0.00508); TCP in base x=-562.598 y=-209.149 z=386.725 mm, rx=1.0611 ry=1.434 rz=-1.4284 rad; joints [-17.931, -67.994, 67.87, -1.514, -17.521, 74.201] deg; flange x=-561.361 y=-17.073 z=388.399 mm, rx=1.3408 ry=-0.992 rz=0.9751 rad
    Wait Sleep waitTime=0.5
    Waypoint Waypoint_39: TCP in base x=-578.257 y=-209.17 z=386.718 mm, rx=1.0688 ry=1.4248 rz=-1.4195 rad; joints [-17.457, -65.682, 64.58, -0.587, -17.021, 75] deg; flange x=-576.975 y=-16.996 z=388.345 mm, rx=1.3356 ry=-1.0021 rz=0.9846 rad
    Wait Sleep waitTime=2
  MoveL speed 76.2 mm/s, acceleration 635 mm/s^2 (recalculateMotions=false) feature=Base
    Waypoint cup_cent: TCP in base x=-519.766 y=-203.654 z=340.589 mm, rx=0.7795 ry=1.7327 rz=-1.7212 rad; joints [-19.983, -73.438, 82.009, -10.178, -19.586, 49.619] deg; flange x=-518.65 y=-11.524 z=342.376 mm, rx=1.4756 ry=-0.6638 rz=0.6489 rad
  Wait Sleep waitTime=15
  MoveL speed 101.6 mm/s, acceleration 889 mm/s^2 (recalculateMotions=false) feature=Base
    Waypoint Waypoint_13: TCP in base x=-436.959 y=-211.169 z=340.586 mm, rx=0.6443 ry=1.8476 rz=-1.8343 rad; joints [-22.817, -84.759, 95.679, -12.333, -22.431, 39.42] deg; flange x=-435.8 y=-19.018 z=342.378 mm, rx=1.5143 ry=-0.528 rz=0.5143 rad
    Waypoint floatbox: TCP in base x=-443.866 y=-210.846 z=92.35 mm, rx=0.6443 ry=1.8475 rz=-1.8342 rad; joints [-22.518, -66.853, 114.574, -49.258, -22.107, 39.554] deg; flange x=-442.761 y=-18.654 z=94.145 mm, rx=1.5143 ry=-0.528 rz=0.5143 rad
    Waypoint putdown: TCP in base x=-443.921 y=-210.82 z=88.782 mm, rx=0.6442 ry=1.8478 rz=-1.8344 rad; joints [-22.518, -66.458, 114.709, -49.79, -22.107, 39.556] deg; flange x=-442.761 y=-18.654 z=90.554 mm, rx=1.5143 ry=-0.528 rz=0.5143 rad
    URCap com.ur.urcap.OnRobot.HelloWorldNode data=depthCompensate = false
      | width = 50
      | name = RG2(50)
      | force = 40
  MoveJ speed 40 deg/s, acceleration 60 deg/s^2 (recalculateMotions=false)
    Waypoint Waypoint_1: TCP in base x=-443.908 y=-10.82 z=88.779 mm, rx=0.6442 ry=1.8478 rz=-1.8343 rad; joints [-43.197, -59.385, 102.633, -44.081, -42.778, 38.753] deg; flange x=-442.761 y=181.337 z=90.554 mm, rx=1.5143 ry=-0.528 rz=0.5143 rad
    URCap com.ur.urcap.OnRobot.HelloWorldNode data=depthCompensate = false
      | width = 80
      | name = RG2(80)
      | force = 40
      | payload = 0.0
    Waypoint Waypoint_4: TCP in base x=-656.767 y=229.451 z=223.061 mm, rx=-1.2339 ry=-1.1819 rz=1.2523 rad; joints [-45.441, -78.027, 106.984, -29.795, 44.386, 3.309] deg; flange x=-464.594 y=230.29 z=220.994 mm, rx=1.1686 ry=-1.2202 rz=-1.1759 rad
  MoveL speed 76.2 mm/s, acceleration 254 mm/s^2 (recalculateMotions=false) feature=Base
    Waypoint Waypoint_12: motionParameters(jointSpeed=1.047198 jointAcceleration=1.396263 cartesianSpeed=0.127 cartesianAcceleration=0.508); TCP in base x=-656.789 y=-220.05 z=206.706 mm, rx=-1.2341 ry=-1.1818 rz=1.2524 rad; joints [15.3, -77.576, 109.185, -32.237, 105.124, 2.532] deg; flange x=-464.594 y=-219.294 z=204.611 mm, rx=1.1686 ry=-1.2202 rz=-1.1759 rad
    Waypoint Waypoint_15: motionParameters(jointSpeed=1.047198 jointAcceleration=1.396263 cartesianSpeed=0.0508 cartesianAcceleration=0.254); TCP in base x=-792.933 y=-220.128 z=193.183 mm, rx=-1.234 ry=-1.1819 rz=1.2524 rad; joints [11.577, -61.699, 88.728, -27.646, 101.411, 2.576] deg; flange x=-600.782 y=-219.294 z=191.088 mm, rx=1.1686 ry=-1.2202 rz=-1.1759 rad
    URCap com.ur.urcap.OnRobot.HelloWorldNode data=depthCompensate = false
      | width = 0
      | name = RG2(0)
      | force = 40
    Waypoint Waypoint_16: TCP in base x=-792.959 y=-220.042 z=221.826 mm, rx=-1.2342 ry=-1.182 rz=1.2522 rad; joints [11.578, -63.351, 86.644, -23.909, 101.41, 2.581] deg; flange x=-600.782 y=-219.294 z=219.879 mm, rx=1.1686 ry=-1.2202 rz=-1.1759 rad
    Wait Sleep waitTime=1
    Waypoint Waypoint_17: motionParameters(jointSpeed=1.047198 jointAcceleration=1.396263 cartesianSpeed=0.0762 cartesianAcceleration=0.254); TCP in base x=-798.941 y=6.682 z=221.951 mm, rx=-1.234 ry=-1.1819 rz=1.2524 rad; joints [-13.021, -68.147, 93.785, -26.25, 76.809, 2.843] deg; flange x=-606.774 y=7.506 z=219.879 mm, rx=1.1686 ry=-1.2202 rz=-1.1759 rad
    Waypoint Waypoint_21: motionParameters(jointSpeed=1.047198 jointAcceleration=1.396263 cartesianSpeed=0.0508 cartesianAcceleration=0.254); TCP in base x=-799.337 y=-1.081 z=93.547 mm, rx=-1.234 ry=-1.1819 rz=1.2523 rad; joints [-12.166, -58.308, 100.871, -43.168, 77.675, 2.811] deg; flange x=-607.165 y=-0.313 z=91.504 mm, rx=1.1686 ry=-1.2202 rz=-1.1759 rad
    URCap com.ur.urcap.OnRobot.HelloWorldNode data=depthCompensate = false
      | width = 90
      | name = RG2(90)
      | force = 40
    Waypoint Waypoint_18: motionParameters(jointSpeed=1.047198 jointAcceleration=1.396263 cartesianSpeed=0.0508 cartesianAcceleration=0.508); TCP in base x=-700.127 y=-1.083 z=93.585 mm, rx=-1.2339 ry=-1.1819 rz=1.2523 rad; joints [-15.057, -68.435, 118.09, -50.266, 74.782, 2.833] deg; flange x=-507.978 y=-0.276 z=91.496 mm, rx=1.1686 ry=-1.2202 rz=-1.176 rad
    MoveJ speed 20 deg/s, acceleration 30 deg/s^2 (recalculateMotions=false)
      Waypoint Waypoint_19: motionParameters(jointSpeed=1.047198 jointAcceleration=1.396263 cartesianSpeed=0.1778 cartesianAcceleration=1.2); TCP in base x=-700.157 y=75.655 z=151.125 mm, rx=-1.234 ry=-1.182 rz=1.2523 rad; joints [-25.04, -73.806, 114.206, -41.049, 64.796, 2.963] deg; flange x=-507.978 y=76.516 z=149.087 mm, rx=1.1686 ry=-1.2202 rz=-1.176 rad
      Waypoint Waypoint_22: motionParameters(nextMotionTime=3); TCP in base x=-404.134 y=-131.897 z=146.449 mm, rx=0.0306 ry=2.2007 rz=-2.1866 rad; joints [-34.074, -73.798, 114.211, -41.08, -34.799, 2.965] deg; flange x=-406.788 y=60.236 z=147.62 mm, rx=1.5769 ry=-0.0219 rz=0.0436 rad
      URCap com.ur.urcap.OnRobot.HelloWorldNode data=depthCompensate = false
        | width = 20
        | name = RG2(20)
        | force = 40
      Waypoint Waypoint_25: motionParameters(jointSpeed=1.047198 jointAcceleration=1.396263 cartesianSpeed=0.249758 cartesianAcceleration=1.2); TCP in base x=-315.793 y=31.161 z=99.113 mm, rx=0.0224 ry=-2.2158 rz=2.195 rad; joints [-58.8, -68.323, 115.476, -47.806, -58.377, -1.11] deg; flange x=-314.66 y=223.315 z=100.907 mm, rx=1.5801 ry=0.0158 rz=-0.0251 rad
